{attribute 'linkalways'} 
{attribute 'no_explicit_call' := 'This FB is a CLASS and must be accessed using methods or properties'}
{attribute 'enable_dynamic_creation'}
FUNCTION_BLOCK _ETcVnContainerExportFormat EXTENDS EnumDatatypeBase
VAR
	localData : ETcVnContainerExportFormat;
	activeData : REFERENCE TO ETcVnContainerExportFormat;
	enumBaseDatatype : _UINT(localData);
END_VAR

METHOD PRIVATE AddLocalEnumeration
VAR_INPUT
	Enumeration : T_MAXSTRING;
	Value : ETcVnContainerExportFormat;
END_VAR
AddEnumeration(Enumeration, Value);
END_METHOD

PROPERTY PUBLIC Address : PVOID
GET
Address := ADR(activeData);
END_GET
END_PROPERTY

METHOD PUBLIC ClearReference
VAR_INPUT
END_VAR
activeData REF= localData;
SetBaseDatatypeReference();
END_METHOD

METHOD PUBLIC Clone : I_Datatype
VAR
    pClone : POINTER TO _ETcVnContainerExportFormat;
END_VAR
pClone := __NEW(_ETcVnContainerExportFormat(InitialValue := Value));
Clone := pClone^;
END_METHOD

METHOD FB_init : BOOL
VAR_INPUT
	bInitRetains : BOOL; // if TRUE, the retain variables are initialized (warm start / cold start)
	bInCopyCode : BOOL;  // if TRUE, the instance afterwards gets moved into the copy code (online change)
	InitialValue : ETcVnContainerExportFormat;
END_VAR
localData := InitialValue;
AddBaseDatatype(enumBaseDatatype);
ClearReference();

AddLocalEnumeration('TCVN_CEF_XML', ETcVnContainerExportFormat.TCVN_CEF_XML);
AddLocalEnumeration('TCVN_CEF_XML_SERIALIZED', ETcVnContainerExportFormat.TCVN_CEF_XML_SERIALIZED);
AddLocalEnumeration('TCVN_CEF_CSV', ETcVnContainerExportFormat.TCVN_CEF_CSV);
AddLocalEnumeration('TCVN_CEF_BINARY', ETcVnContainerExportFormat.TCVN_CEF_BINARY);
END_METHOD

PROPERTY PUBLIC Identifier : T_MAXSTRING
GET
Identifier := 'ETcVnContainerExportFormat';
END_GET
END_PROPERTY

METHOD IsEnumeratorValueEqual : BOOL
VAR_INPUT
	Enumerator : I_KeyValueForwardEnumerator;
END_VAR
VAR
	storedValue : ETcVnContainerExportFormat;
END_VAR
IF NOT Enumerator.TryGet(storedValue) THEN
	RETURN;
END_IF

IsEnumeratorValueEqual := storedValue = activeData;
END_METHOD

METHOD PUBLIC MakeReferenceTo
VAR_INPUT
	ReferenceTarget : REFERENCE TO ETcVnContainerExportFormat;
END_VAR
activeData REF= ReferenceTarget;
SetBaseDatatypeReference();
END_METHOD

METHOD PROTECTED SetBaseDatatypeReference
VAR_INPUT
END_VAR
enumBaseDatatype.MakeReferenceTo(activeData);
END_METHOD

PROPERTY PUBLIC Size : UDINT
GET
Size := SIZEOF(activeData);
END_GET
END_PROPERTY

METHOD TryMakeReferenceTo : BOOL
VAR_INPUT
	Target : I_Datatype;
END_VAR
VAR
	targetAsEnum : I_EnumDatatype;
	pTargetData : POINTER TO ETcVnContainerExportFormat;
END_VAR
IF NOT Target.TryResolveAsEnumDatatype(targetAsEnum) THEN
	RETURN;
END_IF

IF targetAsEnum.Identifier <> Identifier THEN
	RETURN;
END_IF

pTargetData := Target.Address;
activeData REF= pTargetData^;
SetBaseDatatypeReference();
TryMakeReferenceTo := TRUE;
END_METHOD

PROPERTY PUBLIC Value : ETcVnContainerExportFormat
GET
Value := activeData;
END_GET
SET
activeData := Value;
END_SET
END_PROPERTY

END_FUNCTION_BLOCK

(* stored: Version 1.1.0.1, ProductVersion 3.1.4024.13
   POU _ETcVnContainerExportFormat: Id {161114ec-0a78-0497-2d32-e3c9c7bc6f14}, SpecialFunc None
   Folder Core: Id {0a8aeb9a-eb1c-0790-04de-44a2fad60946}
   Folder Protected: Id {309f2cbf-bd6a-0e34-2702-1db1e9b16a6f}
   Folder Customize: Id {3e37b75c-b958-006d-0d79-d353ac70f322}
   Folder Constructor: Id {5022722d-6bbb-0648-23d8-d7c1a1af4778}
   Folder Private: Id {a7a9512e-287d-0882-198c-0cbb284d0044}
   Folder Protected: Id {6dbda530-88b5-080b-2b0a-283f2db7a488}
   Method AddLocalEnumeration: Id {49d7ce3e-32e4-0a45-3372-d3a90f928924}
   Property Address: Id {981064b1-781c-089a-1571-5bf6547320a9}
   Get Get: Id {fb8eebd9-8958-01f5-2fe1-8de9192cb9bf}
   Method ClearReference: Id {a0e7975c-9d1c-0c59-0fb2-5593853cedff}
   Method Clone: Id {e16558de-6671-0737-22f4-3472e5e8bb0c}
   Method FB_init: Id {b348fe2a-52aa-018e-1c41-4bc7c93bece6}
   Property Identifier: Id {df759eff-52fe-0a83-33da-109ca3ad5af4}
   Get Get: Id {460fa355-8f6e-0cd4-1d76-e2abce4c6065}
   Method IsEnumeratorValueEqual: Id {4f01c783-a61b-0695-1b70-72af24afe7db}
   Method MakeReferenceTo: Id {3d929b31-db1c-0bba-0d78-9c9975bee059}
   Method SetBaseDatatypeReference: Id {7684d5c1-bd2f-05f5-3a9e-915ace0210ae}
   Property Size: Id {f107c4d0-7624-0cd1-30e7-2b20f87f5db0}
   Get Get: Id {e9709d44-b740-058c-3b46-1a0a93c3078c}
   Method TryMakeReferenceTo: Id {9d51c386-fdb2-05ea-3e7b-56b50b00243c}
   Property Value: Id {a2c142f0-8fdb-0c6d-06a0-054bff69d723}
   Get Get: Id {3fd3d4d6-9864-0da8-3ac6-78c44747f624}
   Set Set: Id {f8d2547b-bd2f-031b-0a8c-75e1111e5d46} *)
